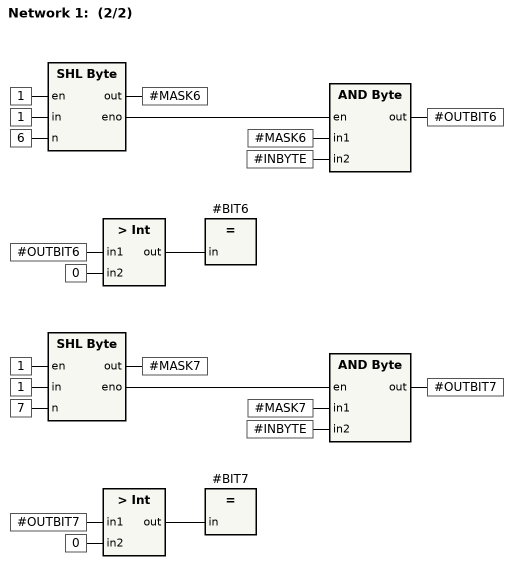
   IF 1 THEN
       #MASK0 := SHL(IN := 1, N := 0);
       #OUTBIT0 := #MASK0 AND #INBYTE;
   END_IF;
   #BIT0 := #OUTBIT0 > 0;
   IF 1 THEN
       #MASK1 := SHL(IN := 1, N := 1);
       #OUTBIT1 := #MASK1 AND #INBYTE;
   END_IF;
   #BIT1 := #OUTBIT1 > 0;
   IF 1 THEN
       #MASK2 := SHL(IN := 1, N := 2);
       #OUTBIT2 := #MASK2 AND #INBYTE;
   END_IF;
   #BIT2 := #OUTBIT2 > 0;
   IF 1 THEN
       #MASK3 := SHL(IN := 1, N := 3);
       #OUTBIT3 := #MASK3 AND #INBYTE;
   END_IF;
   #BIT3 := #OUTBIT3 > 0;
   IF 1 THEN
       #MASK4 := SHL(IN := 1, N := 4);
       #OUTBIT4 := #MASK4 AND #INBYTE;
   END_IF;
   #BIT4 := #OUTBIT4 > 0;
   IF 1 THEN
       #MASK5 := SHL(IN := 1, N := 5);
       #OUTBIT5 := #MASK5 AND #INBYTE;
   END_IF;
   #BIT5 := #OUTBIT5 > 0;
   IF 1 THEN
       #MASK6 := SHL(IN := 1, N := 6);
       #OUTBIT6 := #MASK6 AND #INBYTE;
   END_IF;
   #BIT6 := #OUTBIT6 > 0;
   IF 1 THEN
       #MASK7 := SHL(IN := 1, N := 7);
       #OUTBIT7 := #MASK7 AND #INBYTE;
   END_IF;
   #BIT7 := #OUTBIT7 > 0;
END_REGION
END_FUNCTION

FUNCTION "MOVE_ALMACEN_AUTO" : Void   // FC5, LAD
{ S7_Optimized_Access := 'TRUE' }
VERSION : 0.1
   VAR_INPUT
      STARTF : Bool;
      STOPF : Bool;
      STATESF : Bool;
      BUSYXF : Bool;
      BUSYYF : Bool;
      SEN1F : Bool;
      SEN2F : Bool;
      SEN3F : Bool;
      BIT0XINF : Bool;
      BIT1XINF : Bool;
      BIT2XINF : Bool;
      BIT3XINF : Bool;
      BIT0YINF : Bool;
      BIT1YINF : Bool;
      BIT2YINF : Bool;
      BIT3YINF : Bool;
   END_VAR
   VAR_OUTPUT
      ALARMF : Bool;
      VALVEZF : Bool;
      PINZAF : Bool;
      STATUS2SENDF : Bool;
      STOPXYF : Bool;
      BIT0XOUTF : Bool;
      BIT1XOUTF : Bool;
      BIT2XOUTF : Bool;
      BIT3XOUTF : Bool;
      BIT0YOUTF : Bool;
      BIT1YOUTF : Bool;
      BIT2YOUTF : Bool;
      BIT3YOUTF : Bool;
   END_VAR
   VAR_IN_OUT
      VALXOUTF : Int;
      VALYOUTF : Int;
   END_VAR
   VAR_TEMP
      MEM9F : Bool;
      MEM11F : Bool;
      MEM0F : Bool;
      MEM1F : Bool;
      VALXINF : Int;
      VALYINF : Int;
      MEM2F : Bool;
      MEM3F : Bool;
      MEM4F : Bool;
      MEM5F : Bool;
      MEM6F : Bool;
      MEM7F : Bool;
      MEM8F : Bool;
      MEM10F : Bool;
      MEMYPF : Bool;
      MEMYOF : Bool;
      MEMYP2F : Bool;
      MEMYO2F : Bool;
      ENDPROCESSF : Bool;
      FINF : Bool;
      MEMAUX : Bool;
   END_VAR
   VAR_TEMP   // added for the SCL form of the ladder/FBD networks
      _w1 : Bool;
      _w2 : Bool;
      _w3 : Bool;
      _w4 : Bool;
      _w5 : Bool;
      _w6 : Bool;
      _w7 : Bool;
      _w8 : Bool;
   END_VAR
BEGIN

REGION Network 1: LOGICAL_SEGMENT
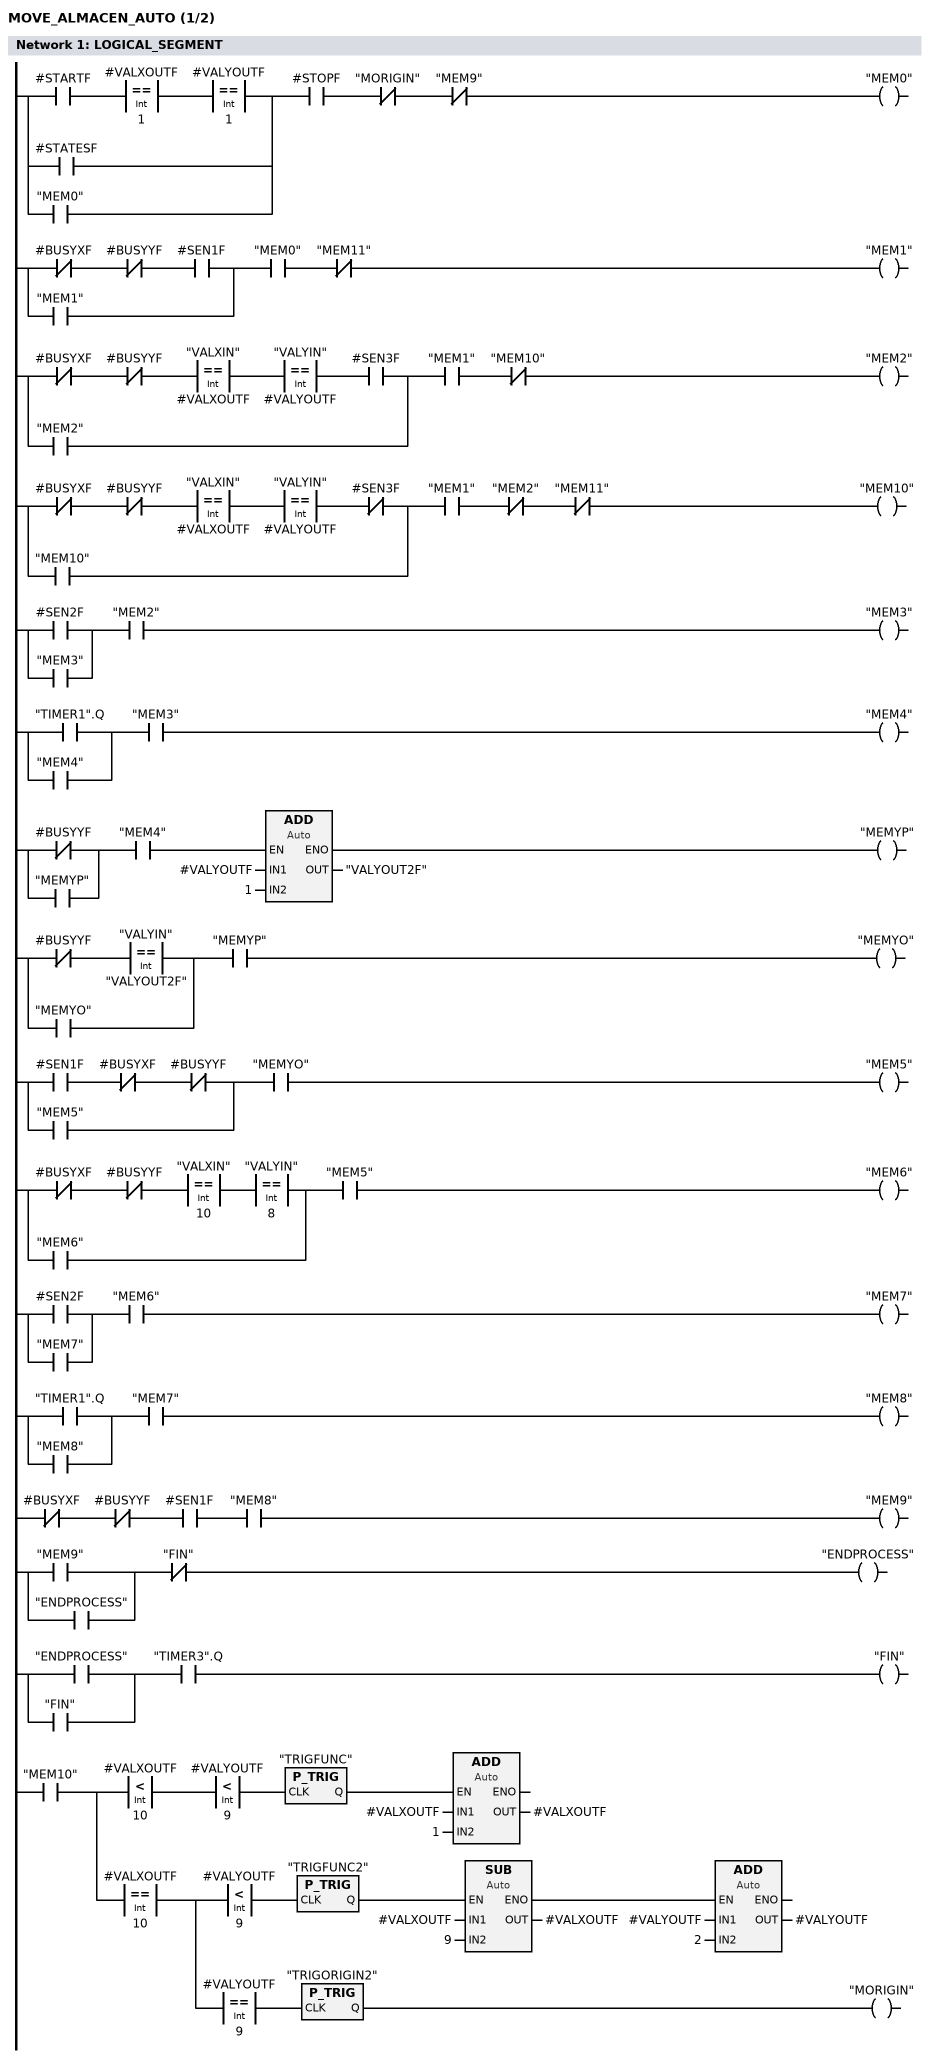
   RUNG wire#powerrail
      Contact( #STARTF )
      { S7_Templates := "SrcType := Int" } EQ_Contact(in1 := #VALXOUTF, in2 := 1)
      { S7_Templates := "SrcType := Int" } EQ_Contact(in1 := #VALYOUTF, in2 := 1)
      wire#w1
      Contact( #STOPF )
      I_Contact( "MORIGIN" )
      I_Contact( "MEM9" )
      Coil( "MEM0" )
   END_RUNG
   RUNG wire#powerrail
      Contact( #STATESF )
   END_RUNG wire#w1
   RUNG wire#powerrail
      Contact( "MEM0" )
   END_RUNG wire#w1
   RUNG wire#powerrail
      I_Contact( #BUSYXF )
      I_Contact( #BUSYYF )
      Contact( #SEN1F )
      wire#w2
      Contact( "MEM0" )
      I_Contact( "MEM11" )
      Coil( "MEM1" )
   END_RUNG
   RUNG wire#powerrail
      Contact( "MEM1" )
   END_RUNG wire#w2
   RUNG wire#powerrail
      I_Contact( #BUSYXF )
      I_Contact( #BUSYYF )
      { S7_Templates := "SrcType := Int" } EQ_Contact(in1 := "VALXIN", in2 := #VALXOUTF)
      { S7_Templates := "SrcType := Int" } EQ_Contact(in1 := "VALYIN", in2 := #VALYOUTF)
      Contact( #SEN3F )
      wire#w3
      Contact( "MEM1" )
      I_Contact( "MEM10" )
      Coil( "MEM2" )
   END_RUNG
   RUNG wire#powerrail
      Contact( "MEM2" )
   END_RUNG wire#w3
   RUNG wire#powerrail
      I_Contact( #BUSYXF )
      I_Contact( #BUSYYF )
      { S7_Templates := "SrcType := Int" } EQ_Contact(in1 := "VALXIN", in2 := #VALXOUTF)
      { S7_Templates := "SrcType := Int" } EQ_Contact(in1 := "VALYIN", in2 := #VALYOUTF)
      I_Contact( #SEN3F )
      wire#w4
      Contact( "MEM1" )
      I_Contact( "MEM2" )
      I_Contact( "MEM11" )
      Coil( "MEM10" )
   END_RUNG
   RUNG wire#powerrail
      Contact( "MEM10" )
   END_RUNG wire#w4
   RUNG wire#powerrail
      Contact( #SEN2F )
      wire#w5
      Contact( "MEM2" )
      Coil( "MEM3" )
   END_RUNG
   RUNG wire#powerrail
      Contact( "MEM3" )
   END_RUNG wire#w5
   RUNG wire#powerrail
      Contact( "TIMER1".Q )
      wire#w6
      Contact( "MEM3" )
      Coil( "MEM4" )
   END_RUNG
   RUNG wire#powerrail
      Contact( "MEM4" )
   END_RUNG wire#w6
   RUNG wire#powerrail
      I_Contact( #BUSYYF )
      wire#w7
      Contact( "MEM4" )
      Add(in1 := #VALYOUTF, in2 := 1, out => "VALYOUT2F")
      Coil( "MEMYP" )
   END_RUNG
   RUNG wire#powerrail
      Contact( "MEMYP" )
   END_RUNG wire#w7
   RUNG wire#powerrail
      I_Contact( #BUSYYF )
      { S7_Templates := "SrcType := Int" } EQ_Contact(in1 := "VALYIN", in2 := "VALYOUT2F")
      wire#w8
      Contact( "MEMYP" )
      Coil( "MEMYO" )
   END_RUNG
   RUNG wire#powerrail
      Contact( "MEMYO" )
   END_RUNG wire#w8
   RUNG wire#powerrail
      Contact( #SEN1F )
      I_Contact( #BUSYXF )
      I_Contact( #BUSYYF )
      wire#w9
      Contact( "MEMYO" )
      Coil( "MEM5" )
   END_RUNG
   RUNG wire#powerrail
      Contact( "MEM5" )
   END_RUNG wire#w9
   RUNG wire#powerrail
      I_Contact( #BUSYXF )
      I_Contact( #BUSYYF )
      { S7_Templates := "SrcType := Int" } EQ_Contact(in1 := "VALXIN", in2 := 10)
      { S7_Templates := "SrcType := Int" } EQ_Contact(in1 := "VALYIN", in2 := 8)
      wire#w10
      Contact( "MEM5" )
      Coil( "MEM6" )
   END_RUNG
   RUNG wire#powerrail
      Contact( "MEM6" )
   END_RUNG wire#w10
   RUNG wire#powerrail
      Contact( #SEN2F )
      wire#w11
      Contact( "MEM6" )
      Coil( "MEM7" )
   END_RUNG
   RUNG wire#powerrail
      Contact( "MEM7" )
   END_RUNG wire#w11
   RUNG wire#powerrail
      Contact( "TIMER1".Q )
      wire#w12
      Contact( "MEM7" )
      Coil( "MEM8" )
   END_RUNG
   RUNG wire#powerrail
      Contact( "MEM8" )
   END_RUNG wire#w12
   RUNG wire#powerrail
      I_Contact( #BUSYXF )
      I_Contact( #BUSYYF )
      Contact( #SEN1F )
      Contact( "MEM8" )
      Coil( "MEM9" )
   END_RUNG
   RUNG wire#powerrail
      Contact( "MEM9" )
      wire#w13
      I_Contact( "FIN" )
      Coil( "ENDPROCESS" )
   END_RUNG
   RUNG wire#powerrail
      Contact( "ENDPROCESS" )
   END_RUNG wire#w13
   RUNG wire#powerrail
      Contact( "ENDPROCESS" )
      wire#w14
      Contact( "TIMER3".Q )
      Coil( "FIN" )
   END_RUNG
   RUNG wire#powerrail
      Contact( "FIN" )
   END_RUNG wire#w14
   RUNG wire#powerrail
      Contact( "MEM10" )
      wire#w15
      { S7_Templates := "SrcType := Int" } LT_Contact(in1 := #VALXOUTF, in2 := 10)
      { S7_Templates := "SrcType := Int" } LT_Contact(in1 := #VALYOUTF, in2 := 9)
      P_Trig( "TRIGFUNC" )
      Add(in1 := #VALXOUTF, in2 := 1, out => #VALXOUTF)
   END_RUNG
   RUNG wire#w15
      { S7_Templates := "SrcType := Int" } EQ_Contact(in1 := #VALXOUTF, in2 := 10)
      wire#w16
      { S7_Templates := "SrcType := Int" } LT_Contact(in1 := #VALYOUTF, in2 := 9)
      P_Trig( "TRIGFUNC2" )
      Sub(in1 := #VALXOUTF, in2 := 9, out => #VALXOUTF)
      Add(in1 := #VALYOUTF, in2 := 2, out => #VALYOUTF)
   END_RUNG
   RUNG wire#w16
      { S7_Templates := "SrcType := Int" } EQ_Contact(in1 := #VALYOUTF, in2 := 9)
      P_Trig( "TRIGORIGIN2" )
      Coil( "MORIGIN" )
   END_RUNG
   // the same network as SCL:
   "MEM0" := ((#STARTF AND (#VALXOUTF = 1) AND (#VALYOUTF = 1)) OR #STATESF OR "MEM0") AND #STOPF AND NOT "MORIGIN" AND NOT "MEM9";
   "MEM1" := ((NOT #BUSYXF AND NOT #BUSYYF AND #SEN1F) OR "MEM1") AND "MEM0" AND NOT "MEM11";
   "MEM2" := ((NOT #BUSYXF AND NOT #BUSYYF AND ("VALXIN" = #VALXOUTF) AND ("VALYIN" = #VALYOUTF) AND #SEN3F) OR "MEM2") AND "MEM1" AND NOT "MEM10";
   "MEM10" := ((NOT #BUSYXF AND NOT #BUSYYF AND ("VALXIN" = #VALXOUTF) AND ("VALYIN" = #VALYOUTF) AND NOT #SEN3F) OR "MEM10") AND "MEM1" AND NOT "MEM2" AND NOT "MEM11";
   "MEM3" := (#SEN2F OR "MEM3") AND "MEM2";
   "MEM4" := ("TIMER1".Q OR "MEM4") AND "MEM3";
   #_w1 := (NOT #BUSYYF OR "MEMYP") AND "MEM4";
   IF #_w1 THEN "VALYOUT2F" := #VALYOUTF + 1; END_IF;
   "MEMYP" := #_w1;
   "MEMYO" := ((NOT #BUSYYF AND ("VALYIN" = "VALYOUT2F")) OR "MEMYO") AND "MEMYP";
   "MEM5" := ((#SEN1F AND NOT #BUSYXF AND NOT #BUSYYF) OR "MEM5") AND "MEMYO";
   "MEM6" := ((NOT #BUSYXF AND NOT #BUSYYF AND ("VALXIN" = 10) AND ("VALYIN" = 8)) OR "MEM6") AND "MEM5";
   "MEM7" := (#SEN2F OR "MEM7") AND "MEM6";
   "MEM8" := ("TIMER1".Q OR "MEM8") AND "MEM7";
   "MEM9" := NOT #BUSYXF AND NOT #BUSYYF AND #SEN1F AND "MEM8";
   "ENDPROCESS" := ("MEM9" OR "ENDPROCESS") AND NOT "FIN";
   "FIN" := ("ENDPROCESS" OR "FIN") AND "TIMER3".Q;
   #_w2 := "MEM10" AND (#VALXOUTF < 10) AND (#VALYOUTF < 9);
   #_w3 := #_w2 AND NOT "TRIGFUNC";   // rising edge
   "TRIGFUNC" := #_w2;
   IF #_w3 THEN #VALXOUTF := #VALXOUTF + 1; END_IF;
   #_w4 := "MEM10" AND (#VALXOUTF = 10);
   #_w5 := #_w4 AND (#VALYOUTF < 9);
   #_w6 := #_w5 AND NOT "TRIGFUNC2";   // rising edge
   "TRIGFUNC2" := #_w5;
   IF #_w6 THEN
       #VALXOUTF := #VALXOUTF - 9;
       #VALYOUTF := #VALYOUTF + 2;
   END_IF;
   #_w7 := #_w4 AND (#VALYOUTF = 9);
   #_w8 := #_w7 AND NOT "TRIGORIGIN2";   // rising edge
   "TRIGORIGIN2" := #_w7;
   "MORIGIN" := #_w8;
END_REGION

REGION Network 2: MECHANICAL_SEGMENT
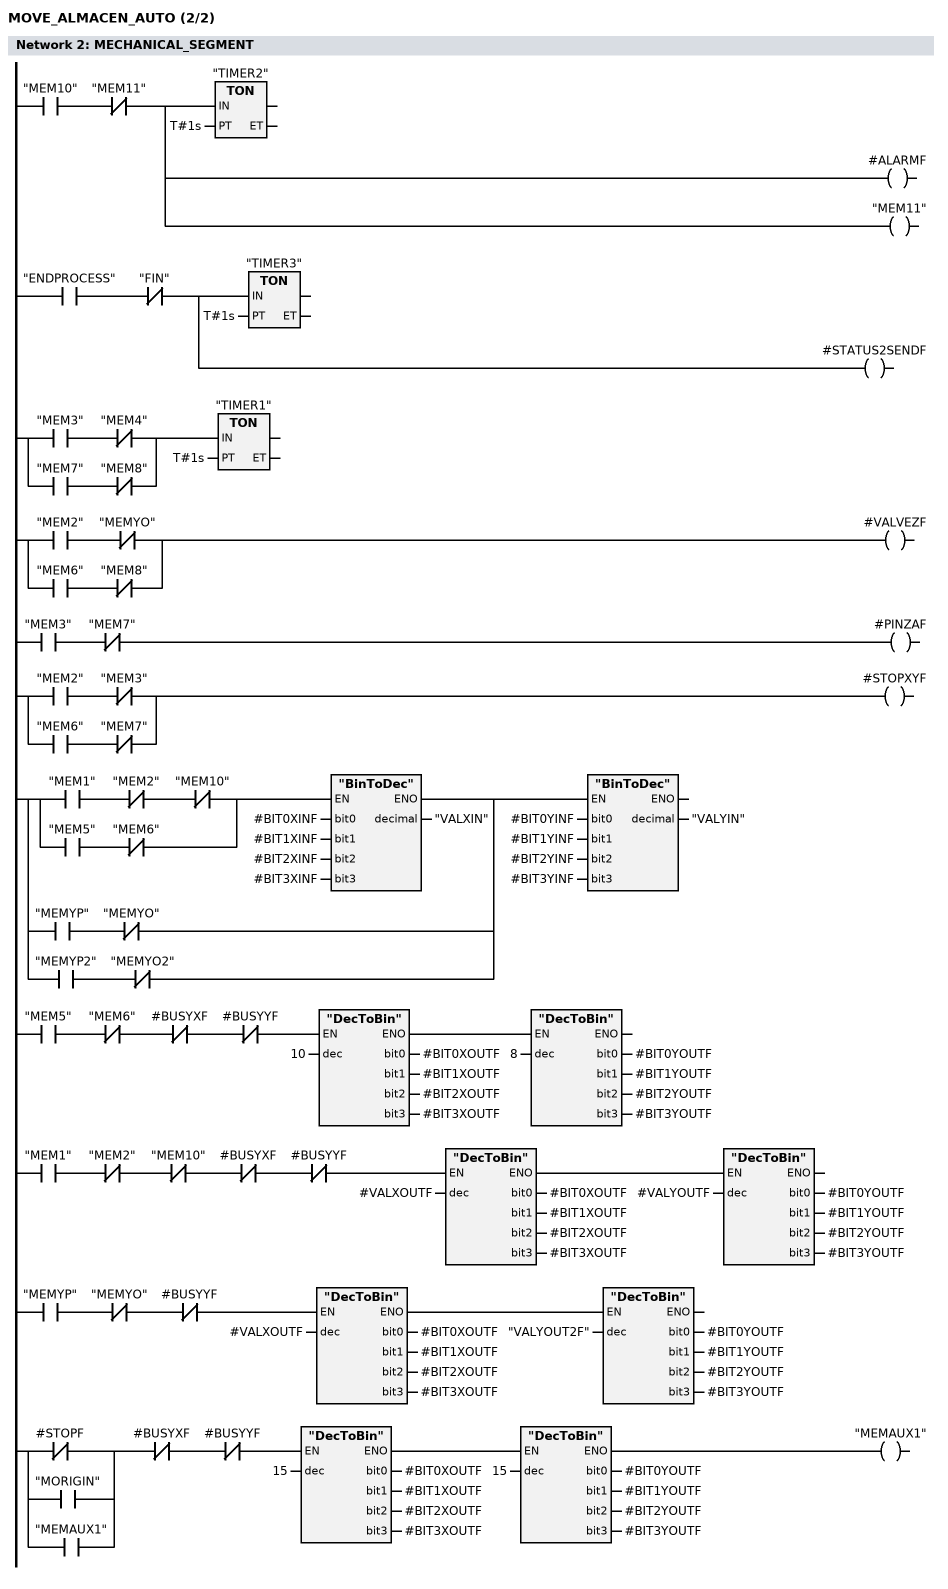
   #_w1 := "MEM10" AND NOT "MEM11";
   "TIMER2".TON(IN := #_w1, PT := T#1s);
   #ALARMF := #_w1;
   "MEM11" := #_w1;
   #_w2 := "ENDPROCESS" AND NOT "FIN";
   "TIMER3".TON(IN := #_w2, PT := T#1s);
   #STATUS2SENDF := #_w2;
   "TIMER1".TON(IN := ("MEM3" AND NOT "MEM4") OR ("MEM7" AND NOT "MEM8"), PT := T#1s);
   #VALVEZF := ("MEM2" AND NOT "MEMYO") OR ("MEM6" AND NOT "MEM8");
   #PINZAF := "MEM3" AND NOT "MEM7";
   #STOPXYF := ("MEM2" AND NOT "MEM3") OR ("MEM6" AND NOT "MEM7");
   "BinToDec"(EN := ("MEM1" AND NOT "MEM2" AND NOT "MEM10") OR ("MEM5" AND NOT "MEM6"),
              bit0 := #BIT0XINF,
              bit1 := #BIT1XINF,
              bit2 := #BIT2XINF,
              bit3 := #BIT3XINF,
              decimal => "VALXIN",
              ENO => #_w3);
   IF #_w3 OR ("MEMYP" AND NOT "MEMYO") OR ("MEMYP2" AND NOT "MEMYO2") THEN
       "BinToDec"(bit0 := #BIT0YINF, bit1 := #BIT1YINF, bit2 := #BIT2YINF, bit3 := #BIT3YINF, decimal => "VALYIN");
   END_IF;
   "DecToBin"(EN := "MEM5" AND NOT "MEM6" AND NOT #BUSYXF AND NOT #BUSYYF,
              dec := 10,
              bit0 => #BIT0XOUTF,
              bit1 => #BIT1XOUTF,
              bit2 => #BIT2XOUTF,
              bit3 => #BIT3XOUTF,
              ENO => #_w4);
   IF #_w4 THEN
       "DecToBin"(dec := 8, bit0 => #BIT0YOUTF, bit1 => #BIT1YOUTF, bit2 => #BIT2YOUTF, bit3 => #BIT3YOUTF);
   END_IF;
   "DecToBin"(EN := "MEM1" AND NOT "MEM2" AND NOT "MEM10" AND NOT #BUSYXF AND NOT #BUSYYF,
              dec := #VALXOUTF,
              bit0 => #BIT0XOUTF,
              bit1 => #BIT1XOUTF,
              bit2 => #BIT2XOUTF,
              bit3 => #BIT3XOUTF,
              ENO => #_w5);
   IF #_w5 THEN
       "DecToBin"(dec := #VALYOUTF, bit0 => #BIT0YOUTF, bit1 => #BIT1YOUTF, bit2 => #BIT2YOUTF, bit3 => #BIT3YOUTF);
   END_IF;
   "DecToBin"(EN := "MEMYP" AND NOT "MEMYO" AND NOT #BUSYYF,
              dec := #VALXOUTF,
              bit0 => #BIT0XOUTF,
              bit1 => #BIT1XOUTF,
              bit2 => #BIT2XOUTF,
              bit3 => #BIT3XOUTF,
              ENO => #_w6);
   IF #_w6 THEN
       "DecToBin"(dec := "VALYOUT2F",
                  bit0 => #BIT0YOUTF,
                  bit1 => #BIT1YOUTF,
                  bit2 => #BIT2YOUTF,
                  bit3 => #BIT3YOUTF);
   END_IF;
   "DecToBin"(EN := (NOT #STOPF OR "MORIGIN" OR "MEMAUX1") AND NOT #BUSYXF AND NOT #BUSYYF,
              dec := 15,
              bit0 => #BIT0XOUTF,
              bit1 => #BIT1XOUTF,
              bit2 => #BIT2XOUTF,
              bit3 => #BIT3XOUTF,
              ENO => #_w7);
   "DecToBin"(EN := #_w7,
              dec := 15,
              bit0 => #BIT0YOUTF,
              bit1 => #BIT1YOUTF,
              bit2 => #BIT2YOUTF,
              bit3 => #BIT3YOUTF,
              ENO => #_w8);
   "MEMAUX1" := #_w8;
END_REGION
END_FUNCTION

FUNCTION "MOVE_ALMACEN" : Void   // FC6, LAD
{ S7_Optimized_Access := 'TRUE' }
VERSION : 0.1
   VAR_INPUT
      STARTF : Bool;
      STOPF : Bool;
      STATESF : Bool;
      BUSYXF : Bool;
      BUSYYF : Bool;
      SEN1F : Bool;
      SEN2F : Bool;
      SEN3F : Bool;
      VALXOUTF : Int;
      VALYOUTF : Int;
      BIT0XINF : Bool;
      BIT1XINF : Bool;
      BIT2XINF : Bool;
      BIT3XINF : Bool;
      BIT0YINF : Bool;
      BIT1YINF : Bool;
      BIT2YINF : Bool;
      BIT3YINF : Bool;
   END_VAR
   VAR_OUTPUT
      ALARMF : Bool;
      VALVEZF : Bool;
      PINZAF : Bool;
      STATUS2SENDF : Bool;
      STOPXYF : Bool;
      BIT0XOUTF : Bool;
      BIT1XOUTF : Bool;
      BIT2XOUTF : Bool;
      BIT3XOUTF : Bool;
      BIT0YOUTF : Bool;
      BIT1YOUTF : Bool;
      BIT2YOUTF : Bool;
      BIT3YOUTF : Bool;
   END_VAR
   VAR_TEMP
      MEM9F : Bool;
      MEM11F : Bool;
      MEM0F : Bool;
      MEM1F : Bool;
      VALXINF : Int;
      VALYINF : Int;
      MEM2F : Bool;
      MEM3F : Bool;
      MEM4F : Bool;
      MEM5F : Bool;
      MEM6F : Bool;
      MEM7F : Bool;
      MEM8F : Bool;
      MEM10F : Bool;
      MEMYPF : Bool;
      MEMYOF : Bool;
      MEMYP2F : Bool;
      MEMYO2F : Bool;
      ENDPROCESSF : Bool;
      FINF : Bool;
      MEMAUX : Bool;
   END_VAR
   VAR_TEMP   // added for the SCL form of the ladder/FBD networks
      _w1 : Bool;
      _w2 : Bool;
      _w3 : Bool;
      _w4 : Bool;
      _w5 : Bool;
      _w6 : Bool;
      _w7 : Bool;
      _w8 : Bool;
   END_VAR
BEGIN

REGION Network 1: LOGICAL_SEGMENT
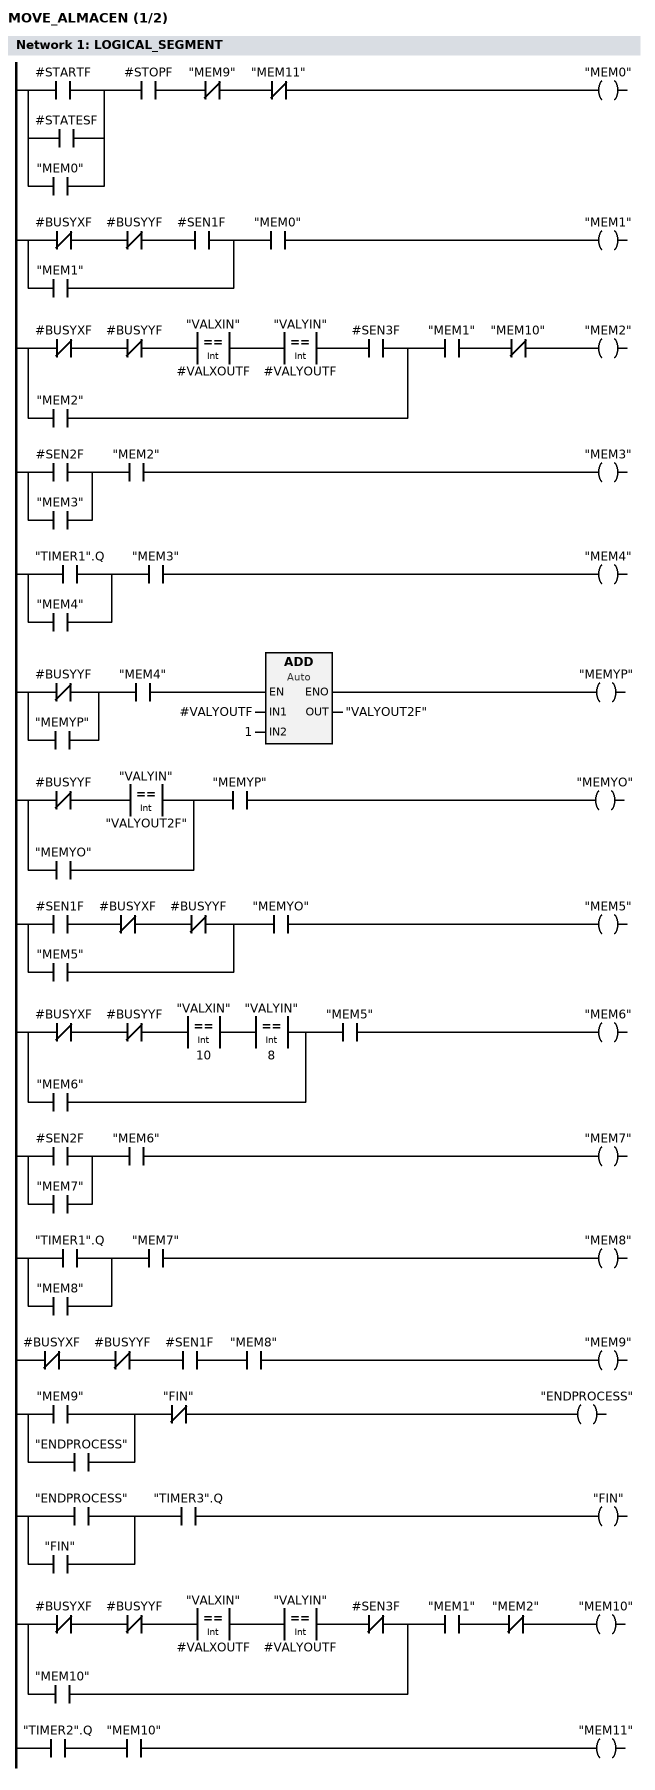
   RUNG wire#powerrail
      Contact( #STARTF )
      wire#w1
      Contact( #STOPF )
      I_Contact( "MEM9" )
      I_Contact( "MEM11" )
      Coil( "MEM0" )
   END_RUNG
   RUNG wire#powerrail
      Contact( #STATESF )
   END_RUNG wire#w1
   RUNG wire#powerrail
      Contact( "MEM0" )
   END_RUNG wire#w1
   RUNG wire#powerrail
      I_Contact( #BUSYXF )
      I_Contact( #BUSYYF )
      Contact( #SEN1F )
      wire#w2
      Contact( "MEM0" )
      Coil( "MEM1" )
   END_RUNG
   RUNG wire#powerrail
      Contact( "MEM1" )
   END_RUNG wire#w2
   RUNG wire#powerrail
      I_Contact( #BUSYXF )
      I_Contact( #BUSYYF )
      { S7_Templates := "SrcType := Int" } EQ_Contact(in1 := "VALXIN", in2 := #VALXOUTF)
      { S7_Templates := "SrcType := Int" } EQ_Contact(in1 := "VALYIN", in2 := #VALYOUTF)
      Contact( #SEN3F )
      wire#w3
      Contact( "MEM1" )
      I_Contact( "MEM10" )
      Coil( "MEM2" )
   END_RUNG
   RUNG wire#powerrail
      Contact( "MEM2" )
   END_RUNG wire#w3
   RUNG wire#powerrail
      Contact( #SEN2F )
      wire#w4
      Contact( "MEM2" )
      Coil( "MEM3" )
   END_RUNG
   RUNG wire#powerrail
      Contact( "MEM3" )
   END_RUNG wire#w4
   RUNG wire#powerrail
      Contact( "TIMER1".Q )
      wire#w5
      Contact( "MEM3" )
      Coil( "MEM4" )
   END_RUNG
   RUNG wire#powerrail
      Contact( "MEM4" )
   END_RUNG wire#w5
   RUNG wire#powerrail
      I_Contact( #BUSYYF )
      wire#w6
      Contact( "MEM4" )
      Add(in1 := #VALYOUTF, in2 := 1, out => "VALYOUT2F")
      Coil( "MEMYP" )
   END_RUNG
   RUNG wire#powerrail
      Contact( "MEMYP" )
   END_RUNG wire#w6
   RUNG wire#powerrail
      I_Contact( #BUSYYF )
      { S7_Templates := "SrcType := Int" } EQ_Contact(in1 := "VALYIN", in2 := "VALYOUT2F")
      wire#w7
      Contact( "MEMYP" )
      Coil( "MEMYO" )
   END_RUNG
   RUNG wire#powerrail
      Contact( "MEMYO" )
   END_RUNG wire#w7
   RUNG wire#powerrail
      Contact( #SEN1F )
      I_Contact( #BUSYXF )
      I_Contact( #BUSYYF )
      wire#w8
      Contact( "MEMYO" )
      Coil( "MEM5" )
   END_RUNG
   RUNG wire#powerrail
      Contact( "MEM5" )
   END_RUNG wire#w8
   RUNG wire#powerrail
      I_Contact( #BUSYXF )
      I_Contact( #BUSYYF )
      { S7_Templates := "SrcType := Int" } EQ_Contact(in1 := "VALXIN", in2 := 10)
      { S7_Templates := "SrcType := Int" } EQ_Contact(in1 := "VALYIN", in2 := 8)
      wire#w9
      Contact( "MEM5" )
      Coil( "MEM6" )
   END_RUNG
   RUNG wire#powerrail
      Contact( "MEM6" )
   END_RUNG wire#w9
   RUNG wire#powerrail
      Contact( #SEN2F )
      wire#w10
      Contact( "MEM6" )
      Coil( "MEM7" )
   END_RUNG
   RUNG wire#powerrail
      Contact( "MEM7" )
   END_RUNG wire#w10
   RUNG wire#powerrail
      Contact( "TIMER1".Q )
      wire#w11
      Contact( "MEM7" )
      Coil( "MEM8" )
   END_RUNG
   RUNG wire#powerrail
      Contact( "MEM8" )
   END_RUNG wire#w11
   RUNG wire#powerrail
      I_Contact( #BUSYXF )
      I_Contact( #BUSYYF )
      Contact( #SEN1F )
      Contact( "MEM8" )
      Coil( "MEM9" )
   END_RUNG
   RUNG wire#powerrail
      Contact( "MEM9" )
      wire#w12
      I_Contact( "FIN" )
      Coil( "ENDPROCESS" )
   END_RUNG
   RUNG wire#powerrail
      Contact( "ENDPROCESS" )
   END_RUNG wire#w12
   RUNG wire#powerrail
      Contact( "ENDPROCESS" )
      wire#w13
      Contact( "TIMER3".Q )
      Coil( "FIN" )
   END_RUNG
   RUNG wire#powerrail
      Contact( "FIN" )
   END_RUNG wire#w13
   RUNG wire#powerrail
      I_Contact( #BUSYXF )
      I_Contact( #BUSYYF )
      { S7_Templates := "SrcType := Int" } EQ_Contact(in1 := "VALXIN", in2 := #VALXOUTF)
      { S7_Templates := "SrcType := Int" } EQ_Contact(in1 := "VALYIN", in2 := #VALYOUTF)
      I_Contact( #SEN3F )
      wire#w14
      Contact( "MEM1" )
      I_Contact( "MEM2" )
      Coil( "MEM10" )
   END_RUNG
   RUNG wire#powerrail
      Contact( "MEM10" )
   END_RUNG wire#w14
   RUNG wire#powerrail
      Contact( "TIMER2".Q )
      Contact( "MEM10" )
      Coil( "MEM11" )
   END_RUNG
   // the same network as SCL:
   "MEM0" := (#STARTF OR #STATESF OR "MEM0") AND #STOPF AND NOT "MEM9" AND NOT "MEM11";
   "MEM1" := ((NOT #BUSYXF AND NOT #BUSYYF AND #SEN1F) OR "MEM1") AND "MEM0";
   "MEM2" := ((NOT #BUSYXF AND NOT #BUSYYF AND ("VALXIN" = #VALXOUTF) AND ("VALYIN" = #VALYOUTF) AND #SEN3F) OR "MEM2") AND "MEM1" AND NOT "MEM10";
   "MEM3" := (#SEN2F OR "MEM3") AND "MEM2";
   "MEM4" := ("TIMER1".Q OR "MEM4") AND "MEM3";
   #_w1 := (NOT #BUSYYF OR "MEMYP") AND "MEM4";
   IF #_w1 THEN "VALYOUT2F" := #VALYOUTF + 1; END_IF;
   "MEMYP" := #_w1;
   "MEMYO" := ((NOT #BUSYYF AND ("VALYIN" = "VALYOUT2F")) OR "MEMYO") AND "MEMYP";
   "MEM5" := ((#SEN1F AND NOT #BUSYXF AND NOT #BUSYYF) OR "MEM5") AND "MEMYO";
   "MEM6" := ((NOT #BUSYXF AND NOT #BUSYYF AND ("VALXIN" = 10) AND ("VALYIN" = 8)) OR "MEM6") AND "MEM5";
   "MEM7" := (#SEN2F OR "MEM7") AND "MEM6";
   "MEM8" := ("TIMER1".Q OR "MEM8") AND "MEM7";
   "MEM9" := NOT #BUSYXF AND NOT #BUSYYF AND #SEN1F AND "MEM8";
   "ENDPROCESS" := ("MEM9" OR "ENDPROCESS") AND NOT "FIN";
   "FIN" := ("ENDPROCESS" OR "FIN") AND "TIMER3".Q;
   "MEM10" := ((NOT #BUSYXF AND NOT #BUSYYF AND ("VALXIN" = #VALXOUTF) AND ("VALYIN" = #VALYOUTF) AND NOT #SEN3F) OR "MEM10") AND "MEM1" AND NOT "MEM2";
   "MEM11" := "TIMER2".Q AND "MEM10";
END_REGION

REGION Network 2: MECHANICAL_SEGMENT
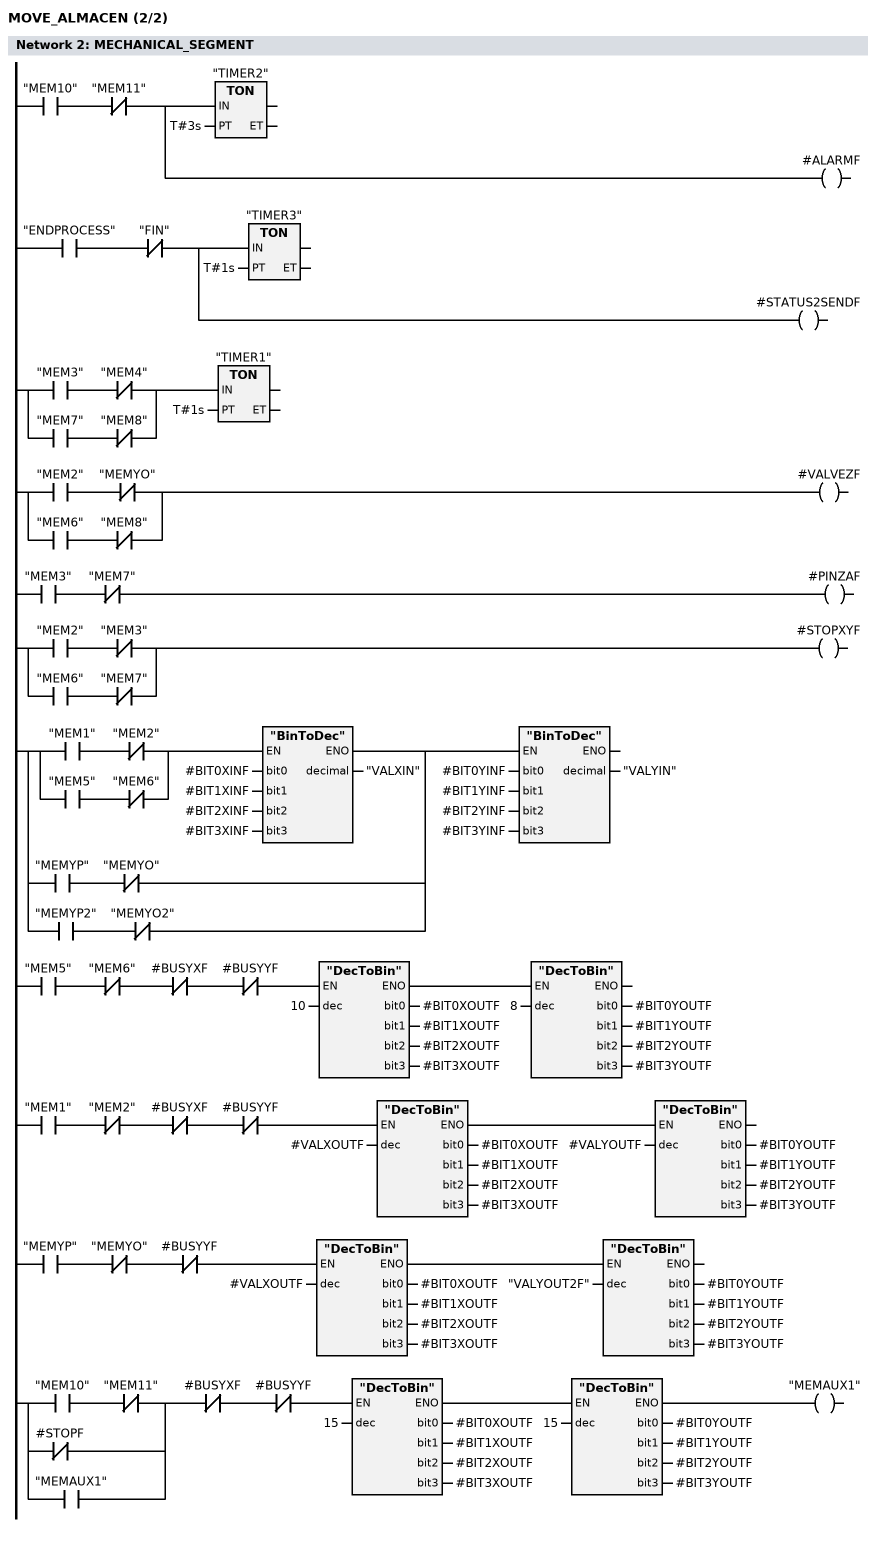
   #_w1 := "MEM10" AND NOT "MEM11";
   "TIMER2".TON(IN := #_w1, PT := T#3s);
   #ALARMF := #_w1;
   #_w2 := "ENDPROCESS" AND NOT "FIN";
   "TIMER3".TON(IN := #_w2, PT := T#1s);
   #STATUS2SENDF := #_w2;
   "TIMER1".TON(IN := ("MEM3" AND NOT "MEM4") OR ("MEM7" AND NOT "MEM8"), PT := T#1s);
   #VALVEZF := ("MEM2" AND NOT "MEMYO") OR ("MEM6" AND NOT "MEM8");
   #PINZAF := "MEM3" AND NOT "MEM7";
   #STOPXYF := ("MEM2" AND NOT "MEM3") OR ("MEM6" AND NOT "MEM7");
   "BinToDec"(EN := ("MEM1" AND NOT "MEM2") OR ("MEM5" AND NOT "MEM6"),
              bit0 := #BIT0XINF,
              bit1 := #BIT1XINF,
              bit2 := #BIT2XINF,
              bit3 := #BIT3XINF,
              decimal => "VALXIN",
              ENO => #_w3);
   IF #_w3 OR ("MEMYP" AND NOT "MEMYO") OR ("MEMYP2" AND NOT "MEMYO2") THEN
       "BinToDec"(bit0 := #BIT0YINF, bit1 := #BIT1YINF, bit2 := #BIT2YINF, bit3 := #BIT3YINF, decimal => "VALYIN");
   END_IF;
   "DecToBin"(EN := "MEM5" AND NOT "MEM6" AND NOT #BUSYXF AND NOT #BUSYYF,
              dec := 10,
              bit0 => #BIT0XOUTF,
              bit1 => #BIT1XOUTF,
              bit2 => #BIT2XOUTF,
              bit3 => #BIT3XOUTF,
              ENO => #_w4);
   IF #_w4 THEN
       "DecToBin"(dec := 8, bit0 => #BIT0YOUTF, bit1 => #BIT1YOUTF, bit2 => #BIT2YOUTF, bit3 => #BIT3YOUTF);
   END_IF;
   "DecToBin"(EN := "MEM1" AND NOT "MEM2" AND NOT #BUSYXF AND NOT #BUSYYF,
              dec := #VALXOUTF,
              bit0 => #BIT0XOUTF,
              bit1 => #BIT1XOUTF,
              bit2 => #BIT2XOUTF,
              bit3 => #BIT3XOUTF,
              ENO => #_w5);
   IF #_w5 THEN
       "DecToBin"(dec := #VALYOUTF, bit0 => #BIT0YOUTF, bit1 => #BIT1YOUTF, bit2 => #BIT2YOUTF, bit3 => #BIT3YOUTF);
   END_IF;
   "DecToBin"(EN := "MEMYP" AND NOT "MEMYO" AND NOT #BUSYYF,
              dec := #VALXOUTF,
              bit0 => #BIT0XOUTF,
              bit1 => #BIT1XOUTF,
              bit2 => #BIT2XOUTF,
              bit3 => #BIT3XOUTF,
              ENO => #_w6);
   IF #_w6 THEN
       "DecToBin"(dec := "VALYOUT2F",
                  bit0 => #BIT0YOUTF,
                  bit1 => #BIT1YOUTF,
                  bit2 => #BIT2YOUTF,
                  bit3 => #BIT3YOUTF);
   END_IF;
   "DecToBin"(EN := (("MEM10" AND NOT "MEM11") OR NOT #STOPF OR "MEMAUX1") AND NOT #BUSYXF AND NOT #BUSYYF,
              dec := 15,
              bit0 => #BIT0XOUTF,
              bit1 => #BIT1XOUTF,
              bit2 => #BIT2XOUTF,
              bit3 => #BIT3XOUTF,
              ENO => #_w7);
   "DecToBin"(EN := #_w7,
              dec := 15,
              bit0 => #BIT0YOUTF,
              bit1 => #BIT1YOUTF,
              bit2 => #BIT2YOUTF,
              bit3 => #BIT3YOUTF,
              ENO => #_w8);
   "MEMAUX1" := #_w8;
END_REGION
END_FUNCTION

ORGANIZATION_BLOCK "Main"   // OB1, LAD, ProgramCycle
TITLE = "Main Program Sweep (Cycle)"
{ S7_Optimized_Access := 'TRUE' }
VERSION : 0.1
   VAR_INPUT
      Initial_Call : Bool;   // Initial call of this OB
      Remanence : Bool;   // =True, if remanent data are available
   END_VAR
   VAR_TEMP
      TIM2 : Time;
      TIM1 : Time;
      MBIT5 : Bool;
      MBIT6 : Bool;
      MBIT3 : Bool;
      MBIT4 : Bool;
      MBIT1 : Bool;
      MBIT2 : Bool;
      MBIT0 : Bool;
   END_VAR
   VAR_TEMP   // added for the SCL form of the ladder/FBD networks
      _w1 : Bool;
      _w2 : Bool;
      _w3 : Bool;
      _w4 : Bool;
      _w5 : Bool;
      _w6 : Bool;
      _w7 : Bool;
      _w8 : Bool;
      _w9 : Bool;
      _w10 : Bool;
   END_VAR
BEGIN

REGION Network 1
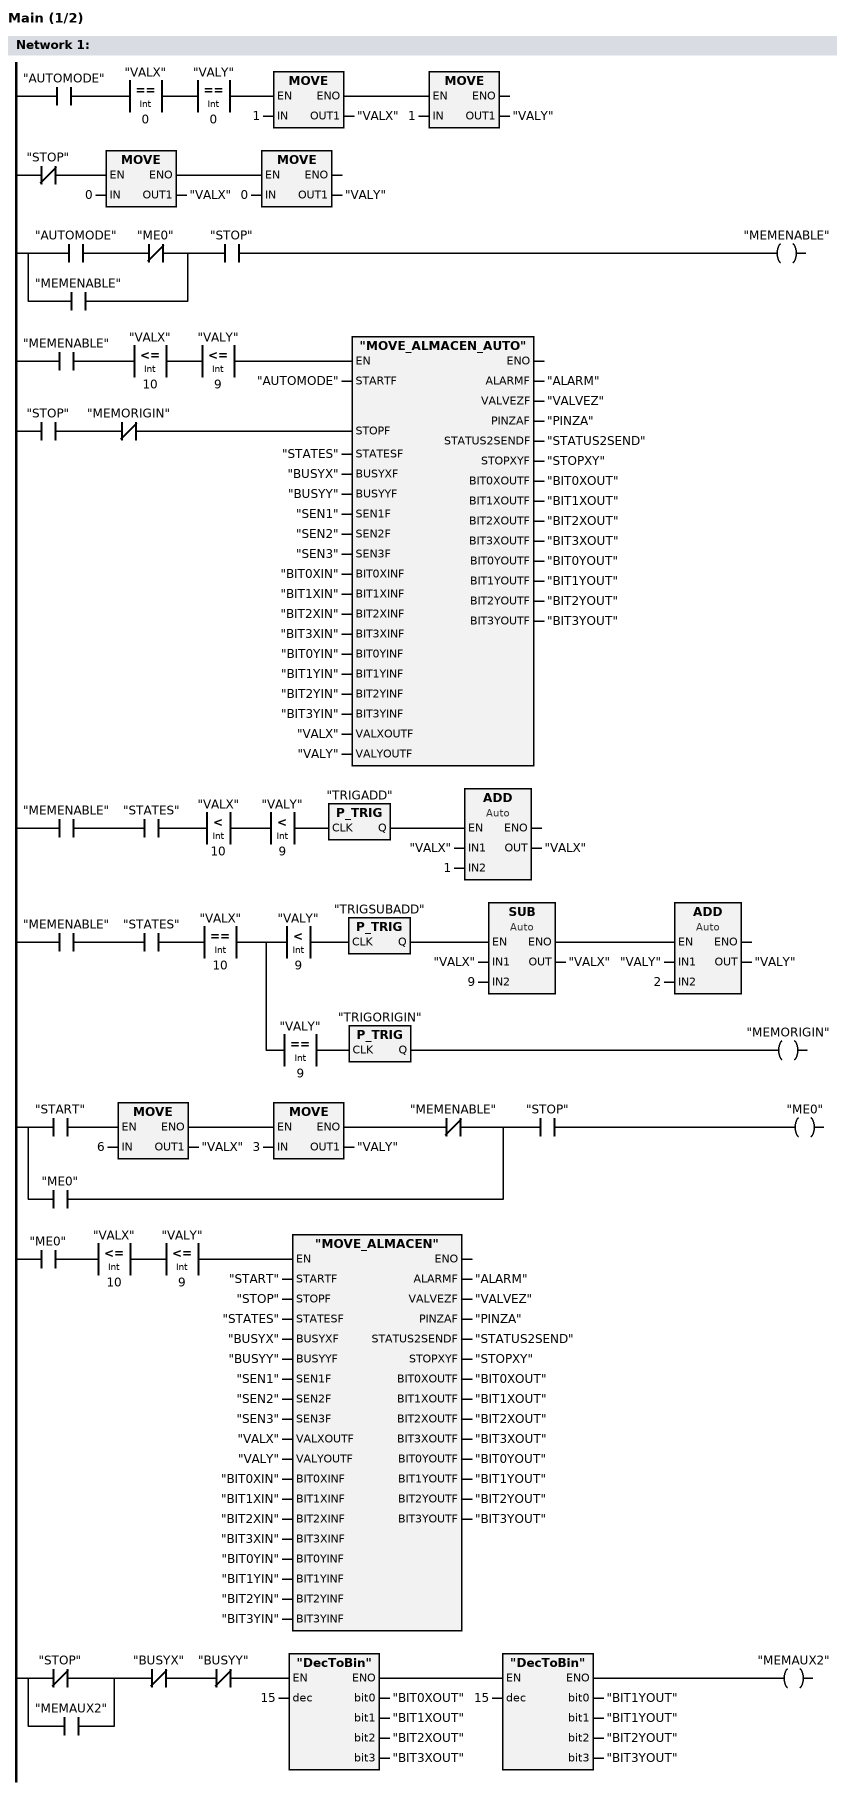
   RUNG wire#powerrail
      Contact( "AUTOMODE" )
      { S7_Templates := "SrcType := Int" } EQ_Contact(in1 := "VALX", in2 := 0)
      { S7_Templates := "SrcType := Int" } EQ_Contact(in1 := "VALY", in2 := 0)
      Move(in := 1, out1 => "VALX")
      Move(in := 1, out1 => "VALY")
   END_RUNG
   RUNG wire#powerrail
      I_Contact( "STOP" )
      Move(in := 0, out1 => "VALX")
      Move(in := 0, out1 => "VALY")
   END_RUNG
   RUNG wire#powerrail
      Contact( "AUTOMODE" )
      I_Contact( "ME0" )
      wire#w1
      Contact( "STOP" )
      Coil( "MEMENABLE" )
   END_RUNG
   RUNG wire#powerrail
      Contact( "MEMENABLE" )
   END_RUNG wire#w1
   RUNG wire#powerrail
      Contact( "MEMENABLE" )
      { S7_Templates := "SrcType := Int" } LE_Contact(in1 := "VALX", in2 := 10)
      { S7_Templates := "SrcType := Int" } LE_Contact(in1 := "VALY", in2 := 9)
      "MOVE_ALMACEN_AUTO"(STOPF := wire#w2, STARTF := "AUTOMODE", STATESF := "STATES", BUSYXF := "BUSYX", BUSYYF := "BUSYY", SEN1F := "SEN1", SEN2F := "SEN2", SEN3F := "SEN3", BIT0XINF := "BIT0XIN", BIT1XINF := "BIT1XIN", BIT2XINF := "BIT2XIN", BIT3XINF := "BIT3XIN", BIT0YINF := "BIT0YIN", BIT1YINF := "BIT1YIN", BIT2YINF := "BIT2YIN", BIT3YINF := "BIT3YIN", VALXOUTF := "VALX", VALYOUTF := "VALY", ALARMF => "ALARM", VALVEZF => "VALVEZ", PINZAF => "PINZA", STATUS2SENDF => "STATUS2SEND", STOPXYF => "STOPXY", BIT0XOUTF => "BIT0XOUT", BIT1XOUTF => "BIT1XOUT", BIT2XOUTF => "BIT2XOUT", BIT3XOUTF => "BIT3XOUT", BIT0YOUTF => "BIT0YOUT", BIT1YOUTF => "BIT1YOUT", BIT2YOUTF => "BIT2YOUT", BIT3YOUTF => "BIT3YOUT")
   END_RUNG
   RUNG wire#powerrail
      Contact( "STOP" )
      I_Contact( "MEMORIGIN" )
   END_RUNG wire#w2
   RUNG wire#powerrail
      Contact( "MEMENABLE" )
      Contact( "STATES" )
      { S7_Templates := "SrcType := Int" } LT_Contact(in1 := "VALX", in2 := 10)
      { S7_Templates := "SrcType := Int" } LT_Contact(in1 := "VALY", in2 := 9)
      P_Trig( "TRIGADD" )
      Add(in1 := "VALX", in2 := 1, out => "VALX")
   END_RUNG
   RUNG wire#powerrail
      Contact( "MEMENABLE" )
      Contact( "STATES" )
      { S7_Templates := "SrcType := Int" } EQ_Contact(in1 := "VALX", in2 := 10)
      wire#w3
      { S7_Templates := "SrcType := Int" } LT_Contact(in1 := "VALY", in2 := 9)
      P_Trig( "TRIGSUBADD" )
      Sub(in1 := "VALX", in2 := 9, out => "VALX")
      Add(in1 := "VALY", in2 := 2, out => "VALY")
   END_RUNG
   RUNG wire#w3
      { S7_Templates := "SrcType := Int" } EQ_Contact(in1 := "VALY", in2 := 9)
      P_Trig( "TRIGORIGIN" )
      Coil( "MEMORIGIN" )
   END_RUNG
   RUNG wire#powerrail
      Contact( "START" )
      Move(in := 6, out1 => "VALX")
      Move(in := 3, out1 => "VALY")
      I_Contact( "MEMENABLE" )
      wire#w4
      Contact( "STOP" )
      Coil( "ME0" )
   END_RUNG
   RUNG wire#powerrail
      Contact( "ME0" )
   END_RUNG wire#w4
   RUNG wire#powerrail
      Contact( "ME0" )
      { S7_Templates := "SrcType := Int" } LE_Contact(in1 := "VALX", in2 := 10)
      { S7_Templates := "SrcType := Int" } LE_Contact(in1 := "VALY", in2 := 9)
      "MOVE_ALMACEN"(STARTF := "START", STOPF := "STOP", STATESF := "STATES", BUSYXF := "BUSYX", BUSYYF := "BUSYY", SEN1F := "SEN1", SEN2F := "SEN2", SEN3F := "SEN3", VALXOUTF := "VALX", VALYOUTF := "VALY", BIT0XINF := "BIT0XIN", BIT1XINF := "BIT1XIN", BIT2XINF := "BIT2XIN", BIT3XINF := "BIT3XIN", BIT0YINF := "BIT0YIN", BIT1YINF := "BIT1YIN", BIT2YINF := "BIT2YIN", BIT3YINF := "BIT3YIN", ALARMF => "ALARM", VALVEZF => "VALVEZ", PINZAF => "PINZA", STATUS2SENDF => "STATUS2SEND", STOPXYF => "STOPXY", BIT0XOUTF => "BIT0XOUT", BIT1XOUTF => "BIT1XOUT", BIT2XOUTF => "BIT2XOUT", BIT3XOUTF => "BIT3XOUT", BIT0YOUTF => "BIT0YOUT", BIT1YOUTF => "BIT1YOUT", BIT2YOUTF => "BIT2YOUT", BIT3YOUTF => "BIT3YOUT")
   END_RUNG
   RUNG wire#powerrail
      I_Contact( "STOP" )
      wire#w5
      I_Contact( "BUSYX" )
      I_Contact( "BUSYY" )
      "DecToBin"(dec := 15, bit0 => "BIT0XOUT", bit1 => "BIT1XOUT", bit2 => "BIT2XOUT", bit3 => "BIT3XOUT")
      "DecToBin"(dec := 15, bit0 => "BIT1YOUT", bit1 => "BIT1YOUT", bit2 => "BIT2YOUT", bit3 => "BIT3YOUT")
      Coil( "MEMAUX2" )
   END_RUNG
   RUNG wire#powerrail
      Contact( "MEMAUX2" )
   END_RUNG wire#w5
   // the same network as SCL:
   #_w1 := "AUTOMODE" AND ("VALX" = 0) AND ("VALY" = 0);
   IF #_w1 THEN
       "VALX" := 1;
       "VALY" := 1;
   END_IF;
   IF NOT "STOP" THEN
       "VALX" := 0;
       "VALY" := 0;
   END_IF;
   "MEMENABLE" := (("AUTOMODE" AND NOT "ME0") OR "MEMENABLE") AND "STOP";
   IF "MEMENABLE" AND ("VALX" <= 10) AND ("VALY" <= 9) THEN
       "MOVE_ALMACEN_AUTO"(STARTF := "AUTOMODE",
                           STOPF := "STOP" AND NOT "MEMORIGIN",
                           STATESF := "STATES",
                           BUSYXF := "BUSYX",
                           BUSYYF := "BUSYY",
                           SEN1F := "SEN1",
                           SEN2F := "SEN2",
                           SEN3F := "SEN3",
                           BIT0XINF := "BIT0XIN",
                           BIT1XINF := "BIT1XIN",
                           BIT2XINF := "BIT2XIN",
                           BIT3XINF := "BIT3XIN",
                           BIT0YINF := "BIT0YIN",
                           BIT1YINF := "BIT1YIN",
                           BIT2YINF := "BIT2YIN",
                           BIT3YINF := "BIT3YIN",
                           VALXOUTF := "VALX",
                           VALYOUTF := "VALY",
                           ALARMF => "ALARM",
                           VALVEZF => "VALVEZ",
                           PINZAF => "PINZA",
                           STATUS2SENDF => "STATUS2SEND",
                           STOPXYF => "STOPXY",
                           BIT0XOUTF => "BIT0XOUT",
                           BIT1XOUTF => "BIT1XOUT",
                           BIT2XOUTF => "BIT2XOUT",
                           BIT3XOUTF => "BIT3XOUT",
                           BIT0YOUTF => "BIT0YOUT",
                           BIT1YOUTF => "BIT1YOUT",
                           BIT2YOUTF => "BIT2YOUT",
                           BIT3YOUTF => "BIT3YOUT");
   END_IF;
   #_w2 := "MEMENABLE" AND "STATES" AND ("VALX" < 10) AND ("VALY" < 9);
   #_w3 := #_w2 AND NOT "TRIGADD";   // rising edge
   "TRIGADD" := #_w2;
   IF #_w3 THEN "VALX" := "VALX" + 1; END_IF;
   #_w4 := "MEMENABLE" AND "STATES" AND ("VALX" = 10);
   #_w5 := #_w4 AND ("VALY" < 9);
   #_w6 := #_w5 AND NOT "TRIGSUBADD";   // rising edge
   "TRIGSUBADD" := #_w5;
   IF #_w6 THEN
       "VALX" := "VALX" - 9;
       "VALY" := "VALY" + 2;
   END_IF;
   #_w7 := #_w4 AND ("VALY" = 9);
   #_w8 := #_w7 AND NOT "TRIGORIGIN";   // rising edge
   "TRIGORIGIN" := #_w7;
   "MEMORIGIN" := #_w8;
   IF "START" THEN
       "VALX" := 6;
       "VALY" := 3;
   END_IF;
   "ME0" := (("START" AND NOT "MEMENABLE") OR "ME0") AND "STOP";
   IF "ME0" AND ("VALX" <= 10) AND ("VALY" <= 9) THEN
       "MOVE_ALMACEN"(STARTF := "START",
                      STOPF := "STOP",
                      STATESF := "STATES",
                      BUSYXF := "BUSYX",
                      BUSYYF := "BUSYY",
                      SEN1F := "SEN1",
                      SEN2F := "SEN2",
                      SEN3F := "SEN3",
                      VALXOUTF := "VALX",
                      VALYOUTF := "VALY",
                      BIT0XINF := "BIT0XIN",
                      BIT1XINF := "BIT1XIN",
                      BIT2XINF := "BIT2XIN",
                      BIT3XINF := "BIT3XIN",
                      BIT0YINF := "BIT0YIN",
                      BIT1YINF := "BIT1YIN",
                      BIT2YINF := "BIT2YIN",
                      BIT3YINF := "BIT3YIN",
                      ALARMF => "ALARM",
                      VALVEZF => "VALVEZ",
                      PINZAF => "PINZA",
                      STATUS2SENDF => "STATUS2SEND",
                      STOPXYF => "STOPXY",
                      BIT0XOUTF => "BIT0XOUT",
                      BIT1XOUTF => "BIT1XOUT",
                      BIT2XOUTF => "BIT2XOUT",
                      BIT3XOUTF => "BIT3XOUT",
                      BIT0YOUTF => "BIT0YOUT",
                      BIT1YOUTF => "BIT1YOUT",
                      BIT2YOUTF => "BIT2YOUT",
                      BIT3YOUTF => "BIT3YOUT");
   END_IF;
   "DecToBin"(EN := (NOT "STOP" OR "MEMAUX2") AND NOT "BUSYX" AND NOT "BUSYY",
              dec := 15,
              bit0 => "BIT0XOUT",
              bit1 => "BIT1XOUT",
              bit2 => "BIT2XOUT",
              bit3 => "BIT3XOUT",
              ENO => #_w9);
   "DecToBin"(EN := #_w9,
              dec := 15,
              bit0 => "BIT1YOUT",
              bit1 => "BIT1YOUT",
              bit2 => "BIT2YOUT",
              bit3 => "BIT3YOUT",
              ENO => #_w10);
   "MEMAUX2" := #_w10;
END_REGION

REGION Network 2: CODER
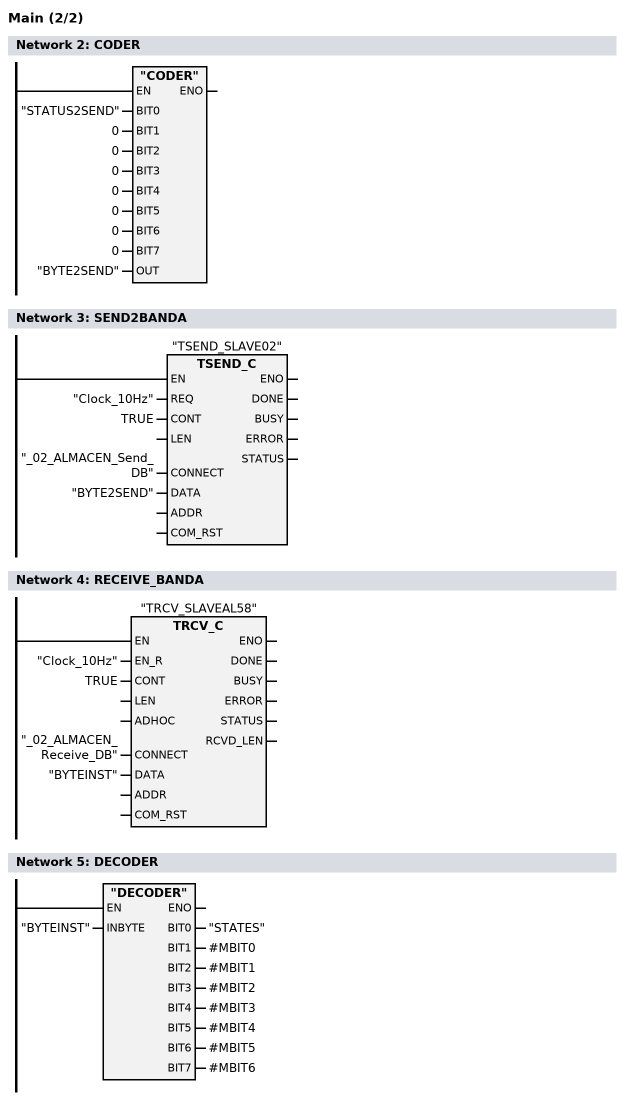
   RUNG wire#powerrail
      "CODER"(BIT0 := "STATUS2SEND", BIT1 := 0, BIT2 := 0, BIT3 := 0, BIT4 := 0, BIT5 := 0, BIT6 := 0, BIT7 := 0, OUT := "BYTE2SEND")
   END_RUNG
   // the same network as SCL:
   "CODER"(BIT0 := "STATUS2SEND",
           BIT1 := 0,
           BIT2 := 0,
           BIT3 := 0,
           BIT4 := 0,
           BIT5 := 0,
           BIT6 := 0,
           BIT7 := 0,
           OUT := "BYTE2SEND");
END_REGION

REGION Network 3: SEND2BANDA
   "TSEND_SLAVE02"(REQ := "Clock_10Hz", CONT := TRUE, CONNECT := "_02_ALMACEN_Send_DB", DATA := "BYTE2SEND");   // TSEND_C
END_REGION

REGION Network 4: RECEIVE_BANDA
   "TRCV_SLAVEAL58"(EN_R := "Clock_10Hz", CONT := TRUE, CONNECT := "_02_ALMACEN_Receive_DB", DATA := "BYTEINST");   // TRCV_C
END_REGION

REGION Network 5: DECODER
   RUNG wire#powerrail
      "DECODER"(INBYTE := "BYTEINST", BIT0 => "STATES", BIT1 => #MBIT0, BIT2 => #MBIT1, BIT3 => #MBIT2, BIT4 => #MBIT3, BIT5 => #MBIT4, BIT6 => #MBIT5, BIT7 => #MBIT6)
   END_RUNG
   // the same network as SCL:
   "DECODER"(INBYTE := "BYTEINST",
             BIT0 => "STATES",
             BIT1 => #MBIT0,
             BIT2 => #MBIT1,
             BIT3 => #MBIT2,
             BIT4 => #MBIT3,
             BIT5 => #MBIT4,
             BIT6 => #MBIT5,
             BIT7 => #MBIT6);
END_REGION
END_ORGANIZATION_BLOCK